FUNCTION_BLOCK FB_BHKW_Modbus
VAR_INPUT
	Adresse				: STRING(15); (* IPv4 address of the target device *)
	BHKW_1_2			: BOOL; (*False = BHKW1, True = BHKW2*)
END_VAR
VAR_OUTPUT
	Zeit_Betrieb		: REAL;	(* h *)
	Zeit_bisWartung		: REAL;	(* h *)
	Temp_Abgas			: REAL;
	Temp_Schallhaube	: REAL;
	Temp_Kuehlwasser	: REAL;
	Temp_Vorlauf		: REAL;
	Temp_Ruecklauf		: REAL;
	Oeldruck			: REAL;	(* bar *)
	Anzahl_Starts		: UINT;
	Leistung_elek		: REAL;
	Drehzahl			: REAL;	(* U/min *)
	Spannung_Generator	: REAL;
	Spannung_Netz		: REAL;
	Strom_Generator		: REAL;
	Frequenz_Netz		: REAL;
	Frequenz_Generator	: REAL;
	CosPHI				: REAL;
	Modul_Modus			: UINT;	(* 0: Aus // 1: Hand // 2: Auto *)
	Modul_Status		: UINT;	(* 0: Aus // 1: Bereit // 2: Start // 3: Betrieb // 4: Störung *)
	Modul_Betriebsart	: UINT;	(* 0: Aus // 1: Hand // 2: Netzersatz // 3:--- // 4: Anwahl 100% // 5: Sollwert 100% *)
	Modul_Meld_Code1	: WORD;	(* Bedeutung s. Datenblatt *)
	Modul_Meld_Code2	: WORD;	(* Bedeutung s. Datenblatt *)
	Modul_Meld_Code3	: WORD;	(* Bedeutung s. Datenblatt *)
	Modul_Meld_Code4	: WORD;	(* Bedeutung s. Datenblatt *)
	Modul_Meld_Code5	: WORD;	(* Bedeutung s. Datenblatt *)
	Modul_Meld_Code6	: WORD;	(* Bedeutung s. Datenblatt *)
	Modul_Meld_Code7	: WORD;	(* Bedeutung s. Datenblatt *)
	Modul_Meld_Code8	: WORD;	(* Bedeutung s. Datenblatt *)
	bReadRegsError_Modus: BOOL;
END_VAR
VAR
	Timer1				: TON;
	Timer2				: TON;
	Timer3				: TON;
	Timer4				: TON;
	Timer5 				: TON;
	Timer6				: TON;
	Timer7				: TON;
	Blinker_Abfrage1		: BOOL;
	Blinker_Abfrage2		: BOOL;
	Blinker_Abfrage3		: BOOL;
	T_on				: TIME:=t#45s;
	T_off				: TIME:=t#10s;
	nSubFnc				: WORD;
	nWriteData			: WORD;
	bDiagnose			: BOOL;
	BHKW_Modul_Modbus: FB_MBReadRegs;
	BHKW_Diagnose		: FB_MBDiagnose;
	Modbus_arrData		: ARRAY  [0..61] OF WORD;
	bDiagnose_busy		: BOOL;
	bDiagnose_Error		: BOOL;
	nDiagnose_ErrorID	: UDINT;
	nRead_Data			: WORD;
	nReadRegsBusy_Modus	: BOOL;
	bReadRegsBusy_Modus	: BOOL;

	nReadRegsErrID_Modus	: UDINT;
	nReadRegsCount_Modus	: UDINT;


	bintest : DWORD:=2#01000010010001111111110011101111;
	realtest: REAL;
	realtest2: REAL;
END_VAR
VAR // added by the converter: edge detectors and wires of the graphical bodies
    _w1, _w3, _w6, _w10, _w14 : REAL;
    _w2 : UINT;
    _w4, _w5, _w7, _w9, _w11, _w13 : ANY;
    _w8, _w12 : BOOL;
END_VAR

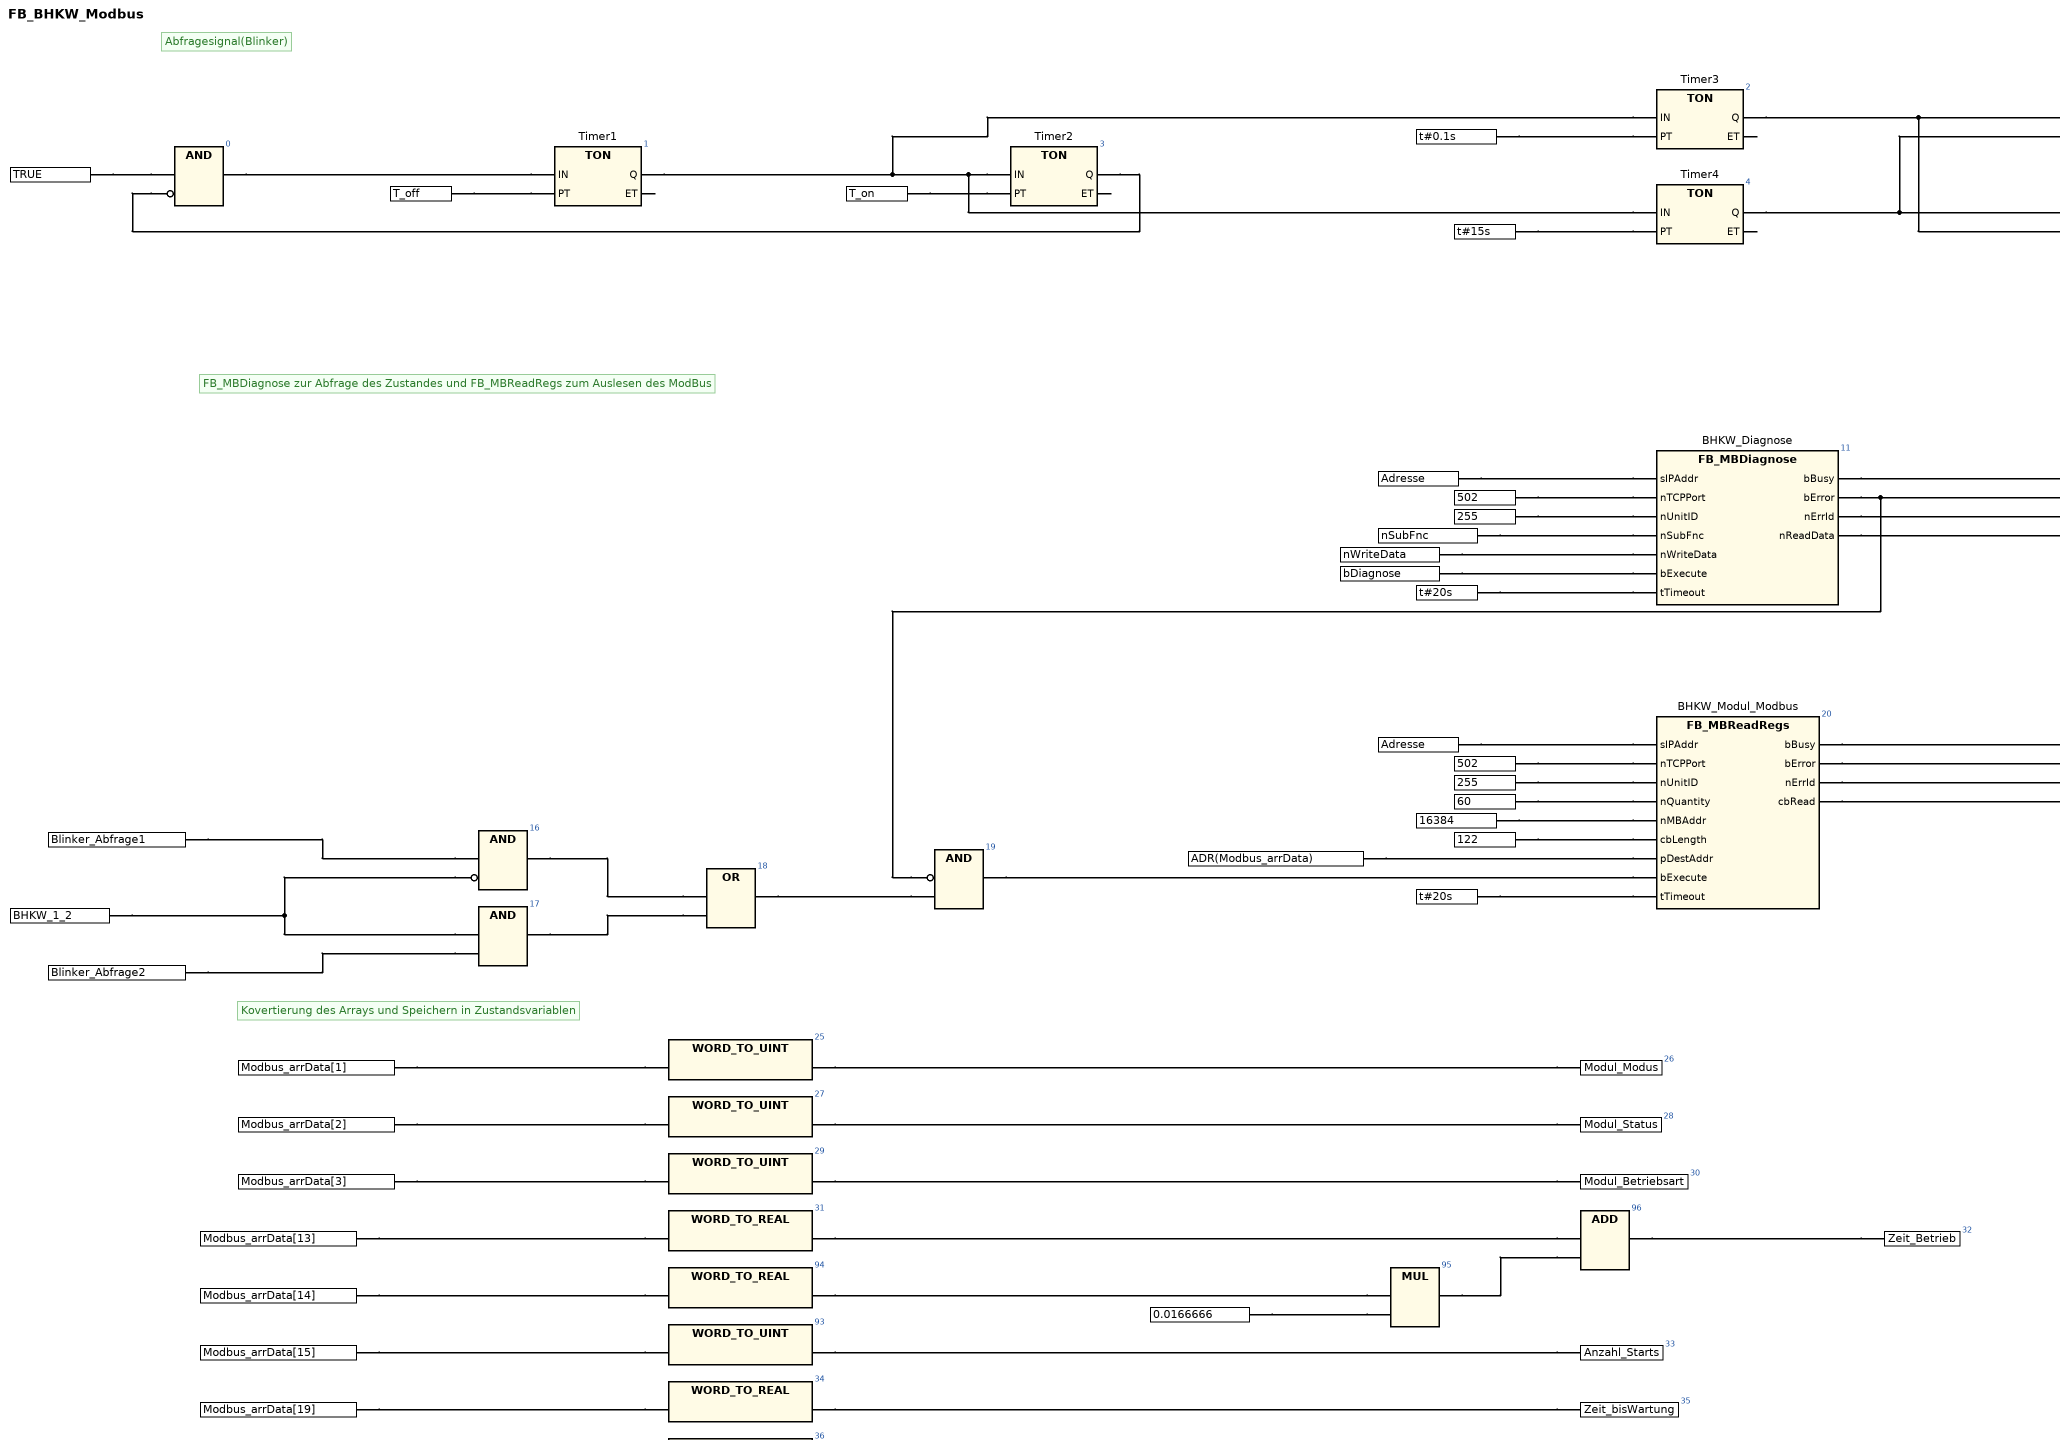
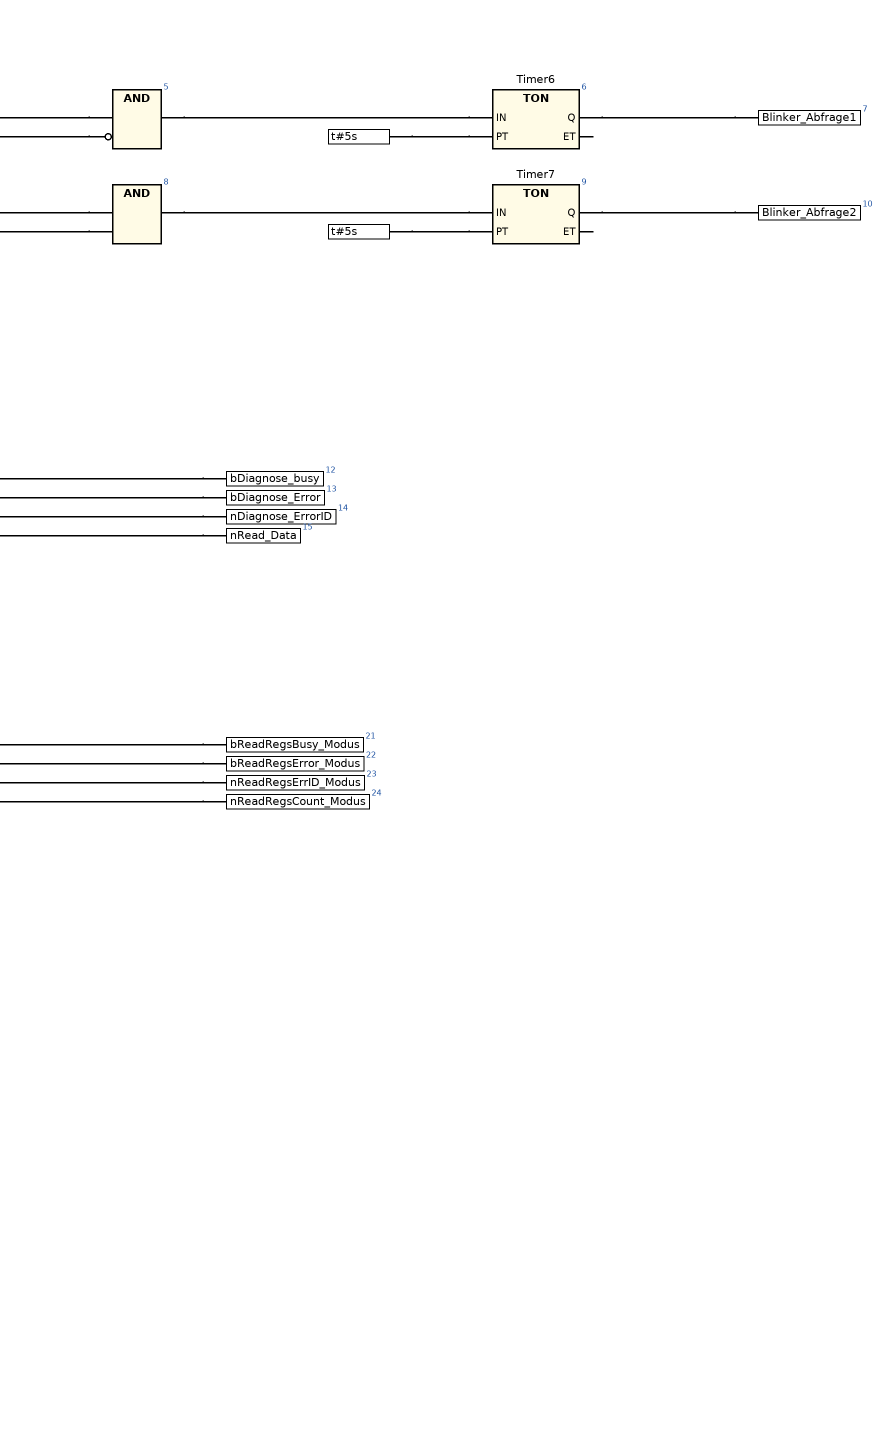
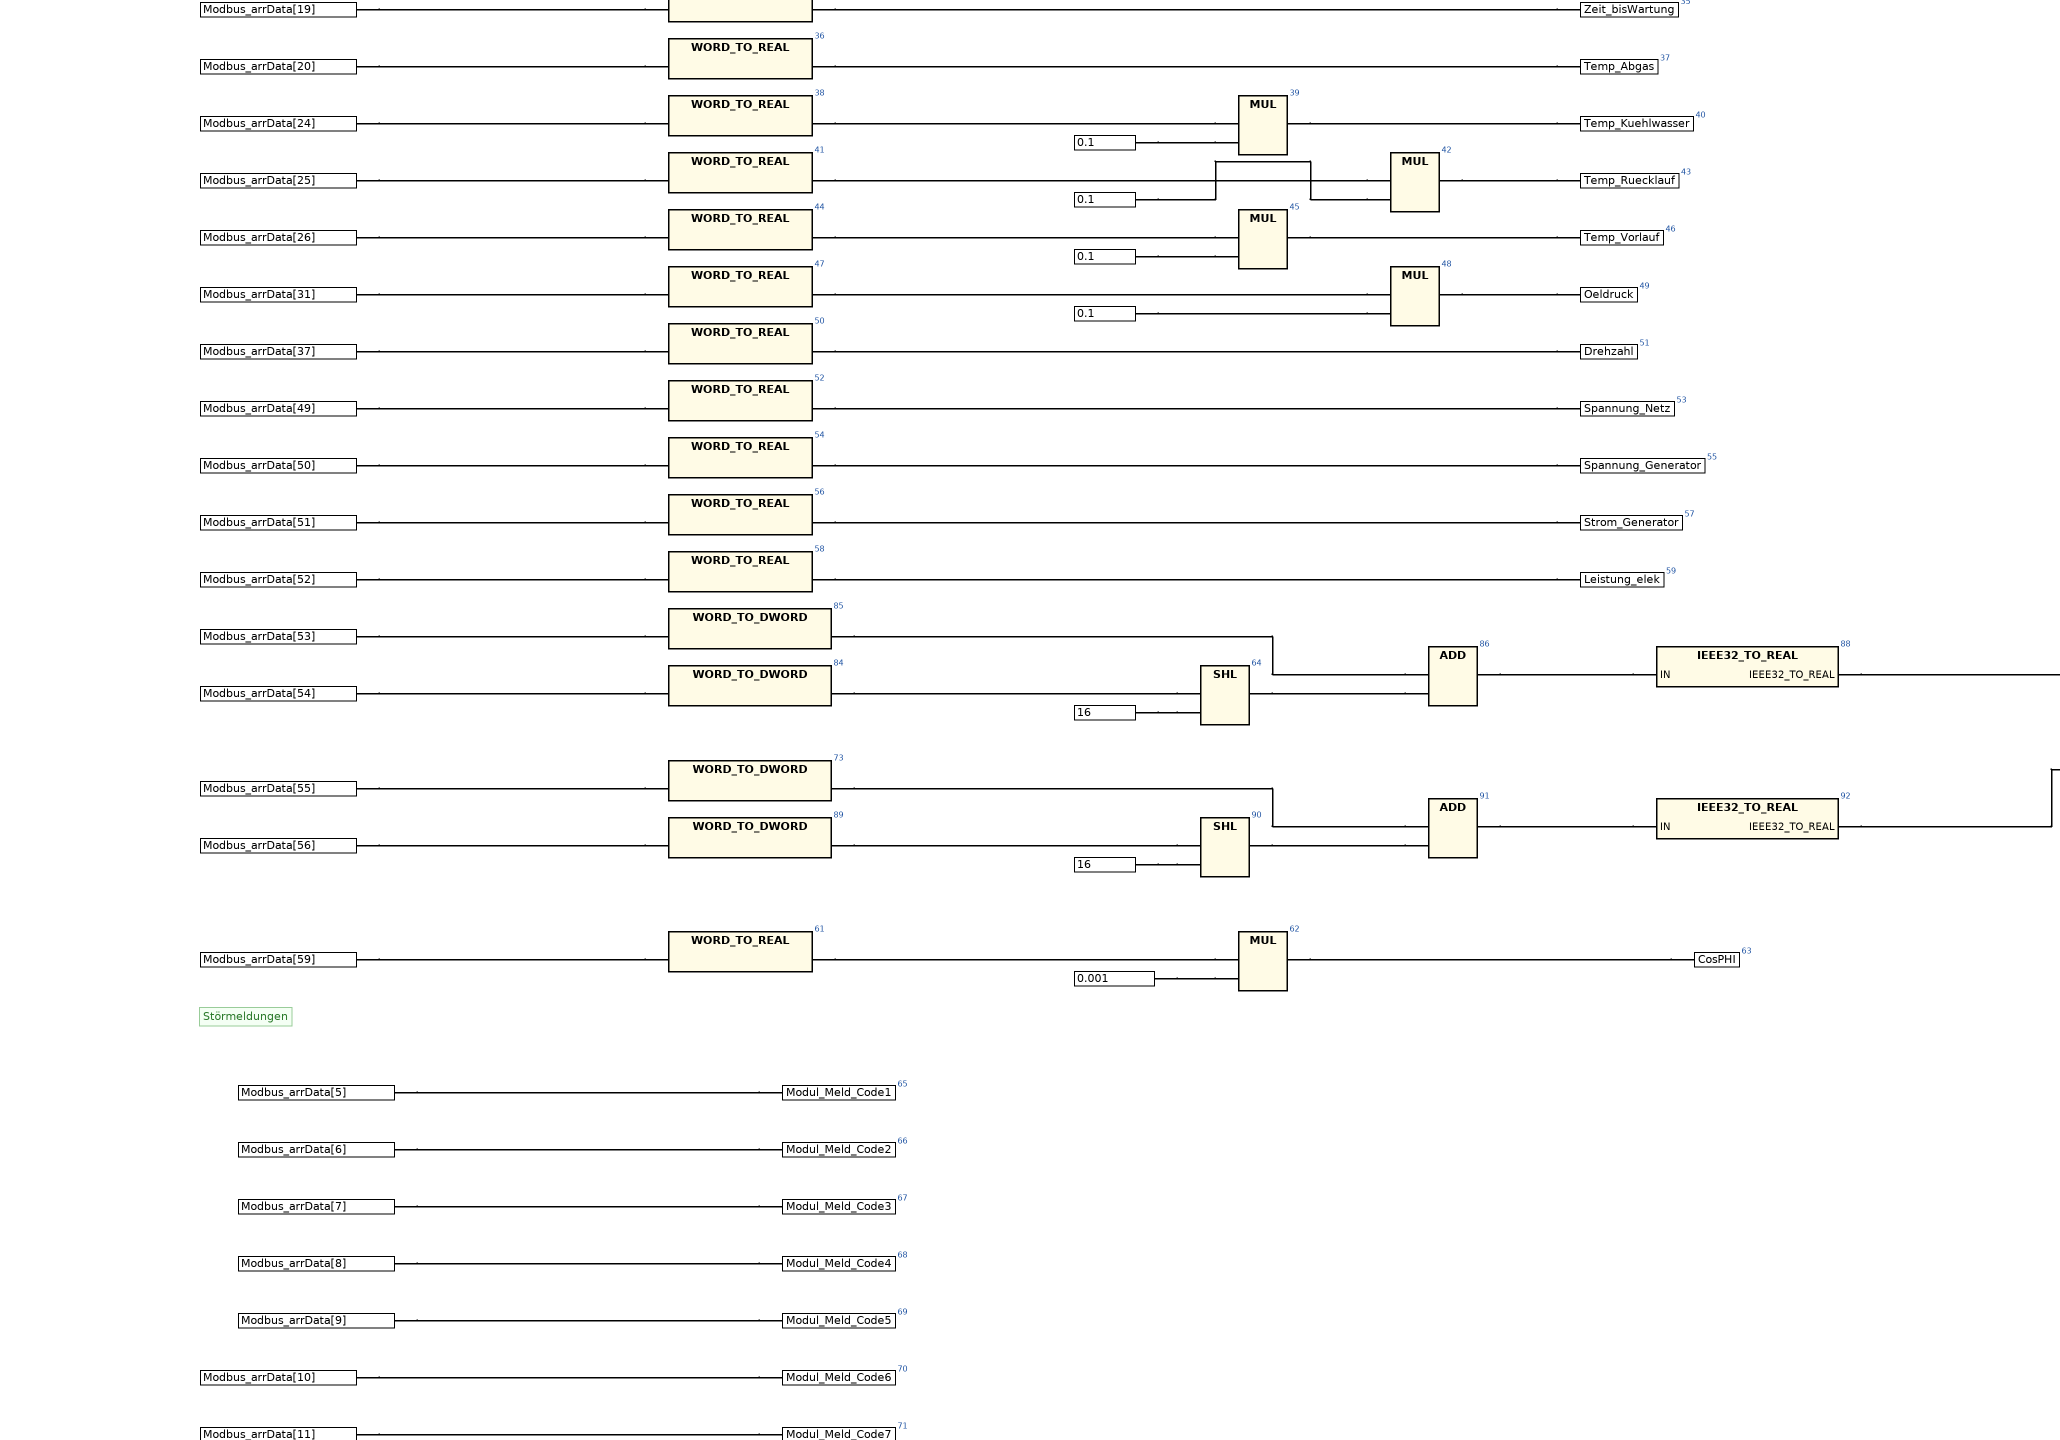
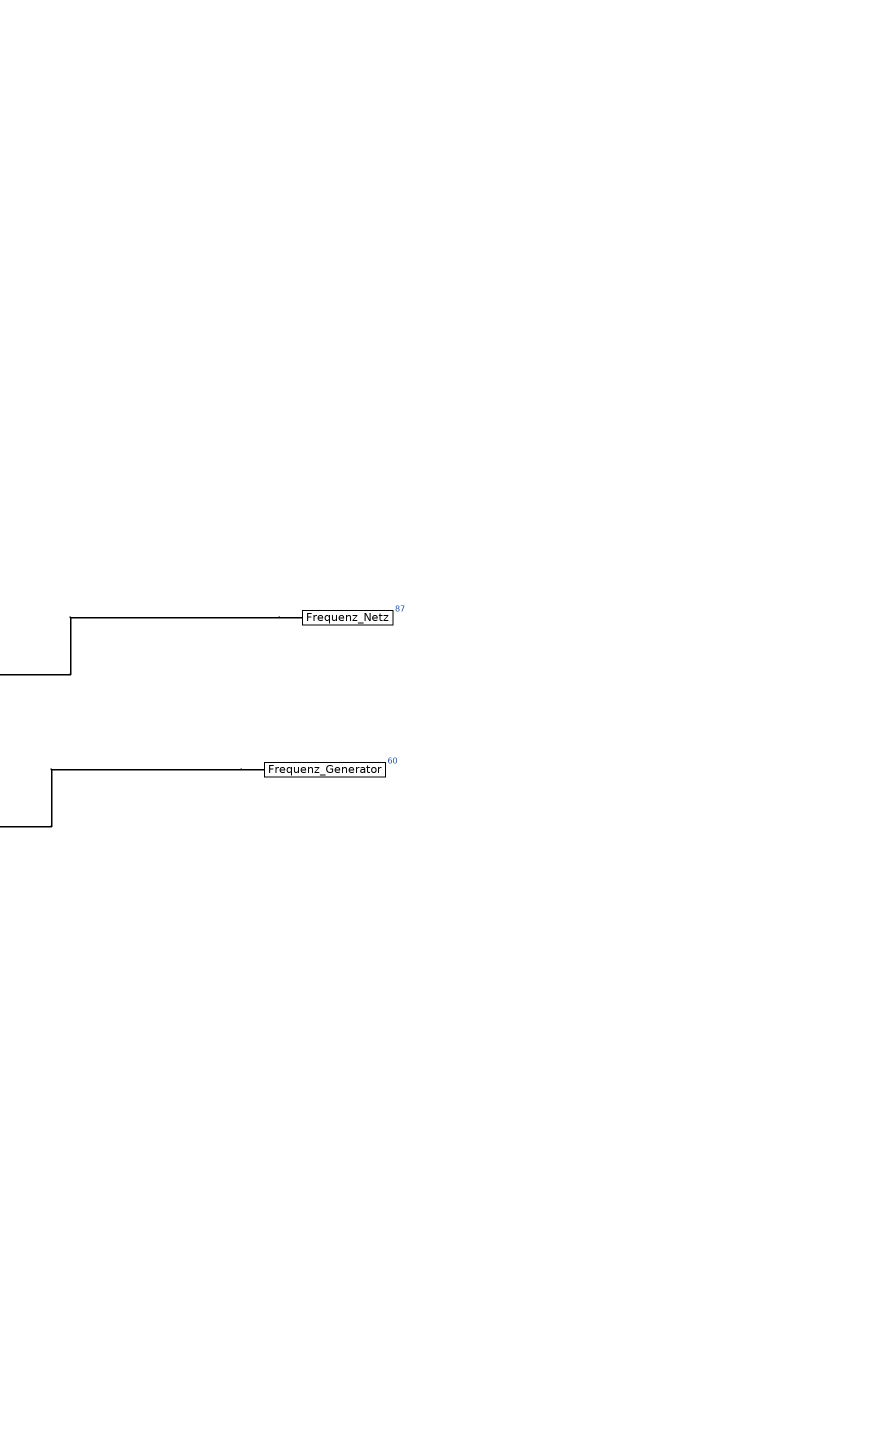
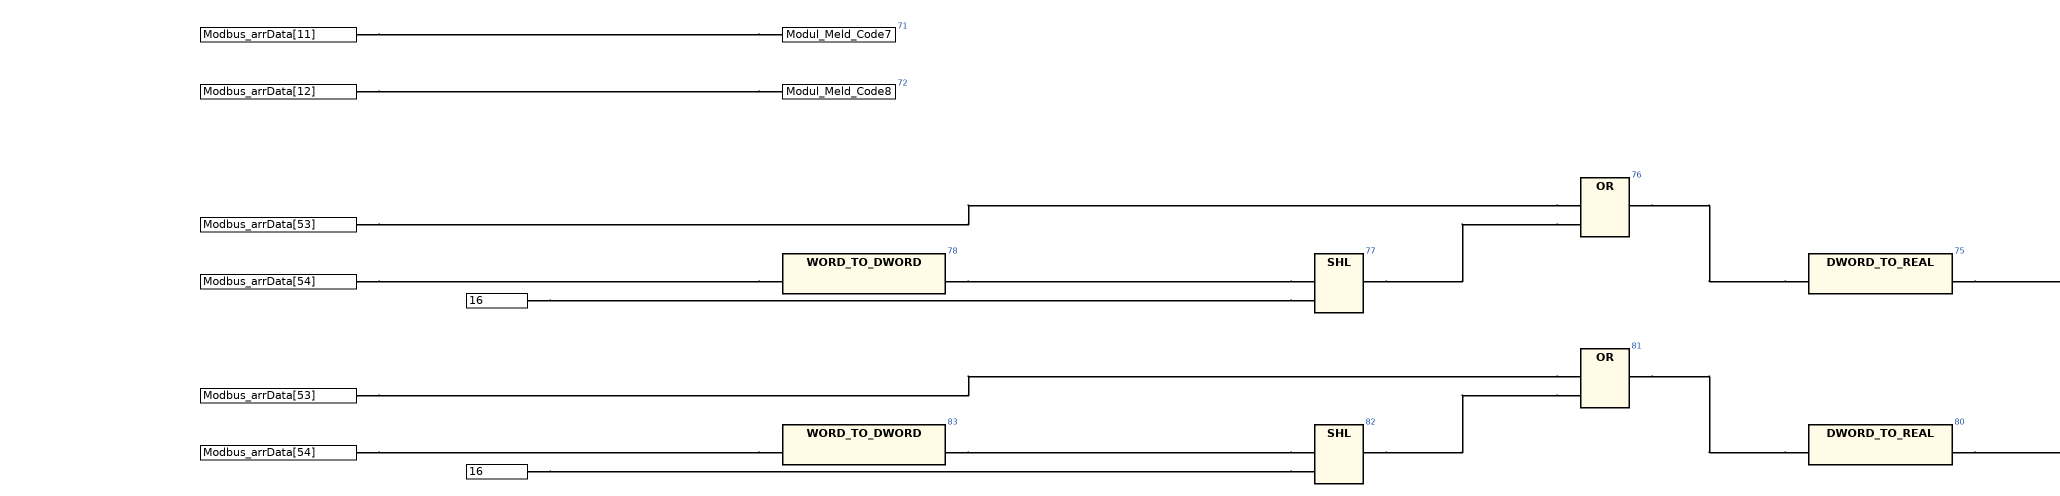
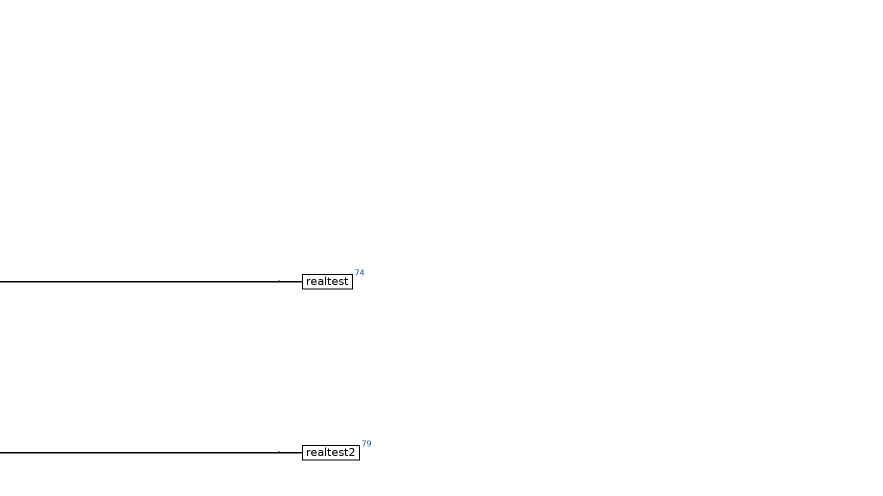
// Abfragesignal(Blinker)
Timer1(IN := TRUE AND NOT Timer2.Q, PT := T_off); // TON
Timer3(IN := Timer1.Q, PT := t#0.1s); // TON
Timer2(IN := Timer1.Q, PT := T_on); // TON
Timer4(IN := Timer1.Q, PT := t#15s); // TON
Timer6(IN := Timer3.Q AND NOT Timer4.Q, PT := t#5s); // TON
Blinker_Abfrage1 := Timer6.Q;
Timer7(IN := Timer4.Q AND Timer3.Q, PT := t#5s); // TON
Blinker_Abfrage2 := Timer7.Q;
BHKW_Diagnose(
    sIPAddr := Adresse,
    nTCPPort := 502,
    nUnitID := 255,
    nSubFnc := nSubFnc,
    nWriteData := nWriteData,
    bExecute := bDiagnose,
    tTimeout := t#20s); // FB_MBDiagnose
bDiagnose_busy := BHKW_Diagnose.bBusy;
bDiagnose_Error := BHKW_Diagnose.bError;
nDiagnose_ErrorID := BHKW_Diagnose.nErrId;
nRead_Data := BHKW_Diagnose.nReadData;
// FB_MBDiagnose zur Abfrage des Zustandes und FB_MBReadRegs zum Auslesen des ModBus
BHKW_Modul_Modbus(
    sIPAddr := Adresse,
    nTCPPort := 502,
    nUnitID := 255,
    nQuantity := 60,
    nMBAddr := 16384,
    cbLength := 122,
    pDestAddr := ADR(Modbus_arrData),
    bExecute := NOT BHKW_Diagnose.bError AND (Blinker_Abfrage1 AND NOT BHKW_1_2 OR BHKW_1_2 AND Blinker_Abfrage2),
    tTimeout := t#20s); // FB_MBReadRegs
bReadRegsBusy_Modus := BHKW_Modul_Modbus.bBusy;
bReadRegsError_Modus := BHKW_Modul_Modbus.bError;
nReadRegsErrID_Modus := BHKW_Modul_Modbus.nErrId;
nReadRegsCount_Modus := BHKW_Modul_Modbus.cbRead;
// Kovertierung des Arrays und Speichern in Zustandsvariablen
Modul_Modus := WORD_TO_UINT(Modbus_arrData[1]);
Modul_Status := WORD_TO_UINT(Modbus_arrData[2]);
Modul_Betriebsart := WORD_TO_UINT(Modbus_arrData[3]);
Zeit_Betrieb := _w1;
Anzahl_Starts := _w2;
Zeit_bisWartung := WORD_TO_REAL(Modbus_arrData[19]);
Temp_Abgas := WORD_TO_REAL(Modbus_arrData[20]);
Temp_Kuehlwasser := WORD_TO_REAL(Modbus_arrData[24]) * 0.1;
Temp_Ruecklauf := WORD_TO_REAL(Modbus_arrData[25]) * 0.1;
Temp_Vorlauf := WORD_TO_REAL(Modbus_arrData[26]) * 0.1;
Oeldruck := WORD_TO_REAL(Modbus_arrData[31]) * 0.1;
Drehzahl := WORD_TO_REAL(Modbus_arrData[37]);
Spannung_Netz := WORD_TO_REAL(Modbus_arrData[49]);
Spannung_Generator := WORD_TO_REAL(Modbus_arrData[50]);
Strom_Generator := WORD_TO_REAL(Modbus_arrData[51]);
Leistung_elek := WORD_TO_REAL(Modbus_arrData[52]);
Frequenz_Generator := _w3;
CosPHI := WORD_TO_REAL(Modbus_arrData[59]) * 0.001;
_w5 := SHL(_w4, 16);
// Störmeldungen
Modul_Meld_Code1 := Modbus_arrData[5];
Modul_Meld_Code2 := Modbus_arrData[6];
Modul_Meld_Code3 := Modbus_arrData[7];
Modul_Meld_Code4 := Modbus_arrData[8];
Modul_Meld_Code5 := Modbus_arrData[9];
Modul_Meld_Code6 := Modbus_arrData[10];
Modul_Meld_Code7 := Modbus_arrData[11];
Modul_Meld_Code8 := Modbus_arrData[12];
realtest := _w6;
_w6 := DWORD_TO_REAL(_w7);
_w7 := Modbus_arrData[53] OR _w8;
_w8 := SHL(_w9, 16);
_w9 := WORD_TO_DWORD(Modbus_arrData[54]);
realtest2 := _w10;
_w10 := DWORD_TO_REAL(_w11);
_w11 := Modbus_arrData[53] OR _w12;
_w12 := SHL(_w13, 16);
_w13 := WORD_TO_DWORD(Modbus_arrData[54]);
_w4 := WORD_TO_DWORD(Modbus_arrData[54]);
Frequenz_Netz := _w14;
_w14 := IEEE32_TO_REAL(IN := WORD_TO_DWORD(Modbus_arrData[53]) + _w5);
_w3 := IEEE32_TO_REAL(IN := WORD_TO_DWORD(Modbus_arrData[55]) + SHL(WORD_TO_DWORD(Modbus_arrData[56]), 16));
_w2 := WORD_TO_UINT(Modbus_arrData[15]);
_w1 := WORD_TO_REAL(Modbus_arrData[13]) + WORD_TO_REAL(Modbus_arrData[14]) * 0.0166666;

END_FUNCTION_BLOCK

(* stored: Version 1.1.0.1, ProductVersion 3.1.4024.9
   POU FB_BHKW_Modbus: Id {ce409556-6322-464d-af4b-a0615e9e20b0}, SpecialFunc None *)
